Staubli VAL3: onStop.pgx

public program onStop(string& x_sItem[])
begin
  if x_sItem=="kill"
    saveProg:libLoad("Disk://kernel/template/session/saveProg/PROG")
    delay(0)
    TrajItem:libLoad("Disk://../templates/trajectory/trajectory.pjx")
    delay(0)
  endIf
end
